// TIA Portal project "Industrial_sorter" (V17)

(* hardware
DEVICE "S7-1500/ET200MP station_1"  S7-1500 station
   slot 0: "Rail_0"  Rack  6ES7 590-1***0-0AA0
   slot 1: "PLC_1"  CPU 1511-1 PN  6ES7 511-1AK00-0AB0  V1.8
      slot 3: "CPU display_1"  6ES7591-1AA00-0AA0
      slot 32768: "PROFINET interface_1"  X1
         slot 32769: "Port_1"  X1 P1
         slot 32770: "Port_2"  X1 P2
*)

// ===== PLC "PLC_1"  CPU 1511-1 PN =====

DATA_BLOCK "Data_block_1"   // DB1
{ S7_Optimized_Access := 'FALSE' }
VERSION : 0.1
   VAR
      Nastro1_run : Bool;
      Fotocellula_ingresso_nastro1 : Bool;
      Val_induttivo : Bool;
      Val_capacitivo : Bool;
      Peso : Real;
      Fotocellula_scan : Bool;
      Fotocellula_ingresso_nastro2 : Bool;
      Tip_oggetto : Int;
      Nastro2_run : Bool;
      Pusher_avanza : Bool;
      Pusher_rientra : Bool;
      Posizione_carrello : Int;
      State_machine : Int;
      Contenitore_target : Int;
      Posizione_target_carrello : Int;
      Posizione_oggetto_X : Real;
      Posizione_oggetto_Y : Real := -1000.0;
      Timer_nastro_ET : DInt;
      Timer_nastro_PT : DInt;
      Sensore_no_oggetti : Bool := false;
      Sistema_START : Bool;
      Sistema_STOP : Bool;
      tempvar1 : Int;
      Contatore : Int;
      Allarme_generale : Bool;
      Allarme_no_tipologia : Bool;
   END_VAR
BEGIN
END_DATA_BLOCK

// folder: System blocks/Program resources

DATA_BLOCK "IEC_Timer_0_DB"   // DB2
{ S7_Optimized_Access := 'TRUE' }
AUTHOR : Simatic
FAMILY : IEC
NAME : IEC_TMR
VERSION : 1.0
// stored: InstanceOfName IEC_TIMER
"IEC_TIMER"
BEGIN
END_DATA_BLOCK

DATA_BLOCK "IEC_Timer_0_DB_1"   // DB3
{ S7_Optimized_Access := 'TRUE' }
AUTHOR : Simatic
FAMILY : IEC
NAME : IEC_TMR
VERSION : 1.0
// stored: InstanceOfName IEC_TIMER
"IEC_TIMER"
BEGIN
END_DATA_BLOCK

DATA_BLOCK "IEC_Timer_0_DB_2"   // DB4
{ S7_Optimized_Access := 'TRUE' }
AUTHOR : Simatic
FAMILY : IEC
NAME : IEC_TMR
VERSION : 1.0
// stored: InstanceOfName IEC_TIMER
"IEC_TIMER"
BEGIN
END_DATA_BLOCK

DATA_BLOCK "IEC_Timer_0_DB_3"   // DB5
{ S7_Optimized_Access := 'TRUE' }
AUTHOR : Simatic
FAMILY : IEC
NAME : IEC_TMR
VERSION : 1.0
// stored: InstanceOfName IEC_TIMER
"IEC_TIMER"
BEGIN
END_DATA_BLOCK

DATA_BLOCK "IEC_Timer_0_DB_4"   // DB6
{ S7_Optimized_Access := 'TRUE' }
AUTHOR : Simatic
FAMILY : IEC
NAME : IEC_TMR
VERSION : 1.0
// stored: InstanceOfName IEC_TIMER
"IEC_TIMER"
BEGIN
END_DATA_BLOCK

DATA_BLOCK "IEC_Timer_0_DB_5"   // DB7
{ S7_Optimized_Access := 'TRUE' }
AUTHOR : Simatic
FAMILY : IEC
NAME : IEC_TMR
VERSION : 1.0
// stored: InstanceOfName IEC_TIMER
"IEC_TIMER"
BEGIN
END_DATA_BLOCK

DATA_BLOCK "IEC_Timer_0_DB_7"   // DB11
{ S7_Optimized_Access := 'TRUE' }
AUTHOR : Simatic
FAMILY : IEC
NAME : IEC_TMR
VERSION : 1.0
// stored: InstanceOfName IEC_TIMER
"IEC_TIMER"
BEGIN
END_DATA_BLOCK

// folder: (top level)

ORGANIZATION_BLOCK "Main"   // OB1, LAD, ProgramCycle
TITLE = "Main Program Sweep (Cycle)"
{ S7_Optimized_Access := 'FALSE' }
VERSION : 0.1
   VAR_TEMP
      EV_CLASS : Byte;   // Bits 0-3 = 1:Coming event, Bits 4-7 = 1:Event class 1
      SCAN_1 : Byte;   // 1:Initial call of the OB, 3: Call 2-n of the OB
      PRIORITY : Byte;   // Priority of OB Execution
      OB_NUMBR : Byte;   // OB number
      RESERVED_1 : Byte;   // Reserved for system
      RESERVED_2 : Byte;   // Reserved for system
      PREV_CYCLE : Int;   // Previous program cycle time (milliseconds)
      MIN_CYCLE : Int;   // Minimum program cycle time (milliseconds)
      MAX_CYCLE : Int;   // Maximum program cycle time (milliseconds)
      DATE_TIME : Date_And_Time;   // Date and time OB started
   END_VAR
   VAR_TEMP   // added for the SCL form of the ladder/FBD networks
      _w1 : Bool;
      _w2 : Bool;
   END_VAR
BEGIN

REGION Network 1
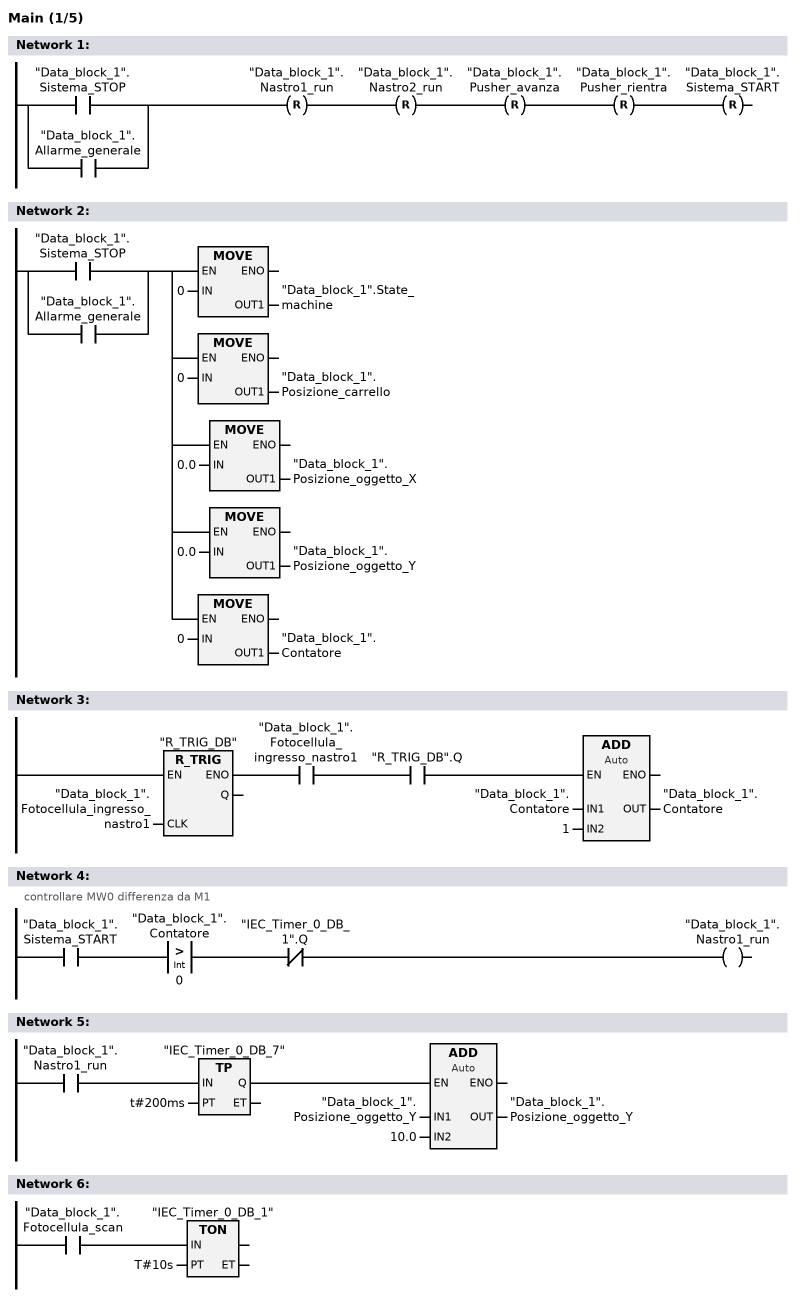
   RUNG wire#powerrail
      Contact( "Data_block_1".Sistema_STOP )
      wire#w1
      R_Coil( "Data_block_1".Nastro1_run )
      R_Coil( "Data_block_1".Nastro2_run )
      R_Coil( "Data_block_1".Pusher_avanza )
      R_Coil( "Data_block_1".Pusher_rientra )
      R_Coil( "Data_block_1".Sistema_START )
   END_RUNG
   RUNG wire#powerrail
      Contact( "Data_block_1".Allarme_generale )
   END_RUNG wire#w1
   // the same network as SCL:
   IF "Data_block_1".Sistema_STOP OR "Data_block_1".Allarme_generale THEN
       "Data_block_1".Nastro1_run := FALSE;
       "Data_block_1".Nastro2_run := FALSE;
       "Data_block_1".Pusher_avanza := FALSE;
       "Data_block_1".Pusher_rientra := FALSE;
       "Data_block_1".Sistema_START := FALSE;
   END_IF;
END_REGION

REGION Network 2
   RUNG wire#powerrail
      Contact( "Data_block_1".Sistema_STOP )
      wire#w1
      Move(in := 0, out1 => "Data_block_1".State_machine)
   END_RUNG
   RUNG wire#powerrail
      Contact( "Data_block_1".Allarme_generale )
   END_RUNG wire#w1
   RUNG wire#w1
      Move(in := 0, out1 => "Data_block_1".Posizione_carrello)
   END_RUNG
   RUNG wire#w1
      Move(in := 0.0, out1 => "Data_block_1".Posizione_oggetto_X)
   END_RUNG
   RUNG wire#w1
      Move(in := 0.0, out1 => "Data_block_1".Posizione_oggetto_Y)
   END_RUNG
   RUNG wire#w1
      Move(in := 0, out1 => "Data_block_1".Contatore)
   END_RUNG
   // the same network as SCL:
   IF "Data_block_1".Sistema_STOP OR "Data_block_1".Allarme_generale THEN
       "Data_block_1".State_machine := 0;
       "Data_block_1".Posizione_carrello := 0;
       "Data_block_1".Posizione_oggetto_X := 0.0;
       "Data_block_1".Posizione_oggetto_Y := 0.0;
       "Data_block_1".Contatore := 0;
   END_IF;
END_REGION

REGION Network 3
   // ENO of a box is taken as its EN; it also drops when the box reports an error
   "R_TRIG_DB"(CLK := "Data_block_1".Fotocellula_ingresso_nastro1);   // R_TRIG
   IF "Data_block_1".Fotocellula_ingresso_nastro1 AND "R_TRIG_DB".Q THEN
       "Data_block_1".Contatore := "Data_block_1".Contatore + 1;
   END_IF;
END_REGION

REGION Network 4
   // controllare MW0 differenza da M1
   RUNG wire#powerrail
      Contact( "Data_block_1".Sistema_START )
      { S7_Templates := "SrcType := Int" } GT_Contact(in1 := "Data_block_1".Contatore, in2 := 0)
      I_Contact( "IEC_Timer_0_DB_1".Q )
      Coil( "Data_block_1".Nastro1_run )
   END_RUNG
   // the same network as SCL:
   "Data_block_1".Nastro1_run := "Data_block_1".Sistema_START AND ("Data_block_1".Contatore > 0) AND NOT "IEC_Timer_0_DB_1".Q;
END_REGION

REGION Network 5
   "IEC_Timer_0_DB_7".TP(IN := "Data_block_1".Nastro1_run, PT := t#200ms);
   IF "IEC_Timer_0_DB_7".Q THEN
       "Data_block_1".Posizione_oggetto_Y := "Data_block_1".Posizione_oggetto_Y + 10.0;
   END_IF;
END_REGION

REGION Network 6
   "IEC_Timer_0_DB_1".TON(IN := "Data_block_1".Fotocellula_scan, PT := T#10s);
END_REGION

REGION Network 7
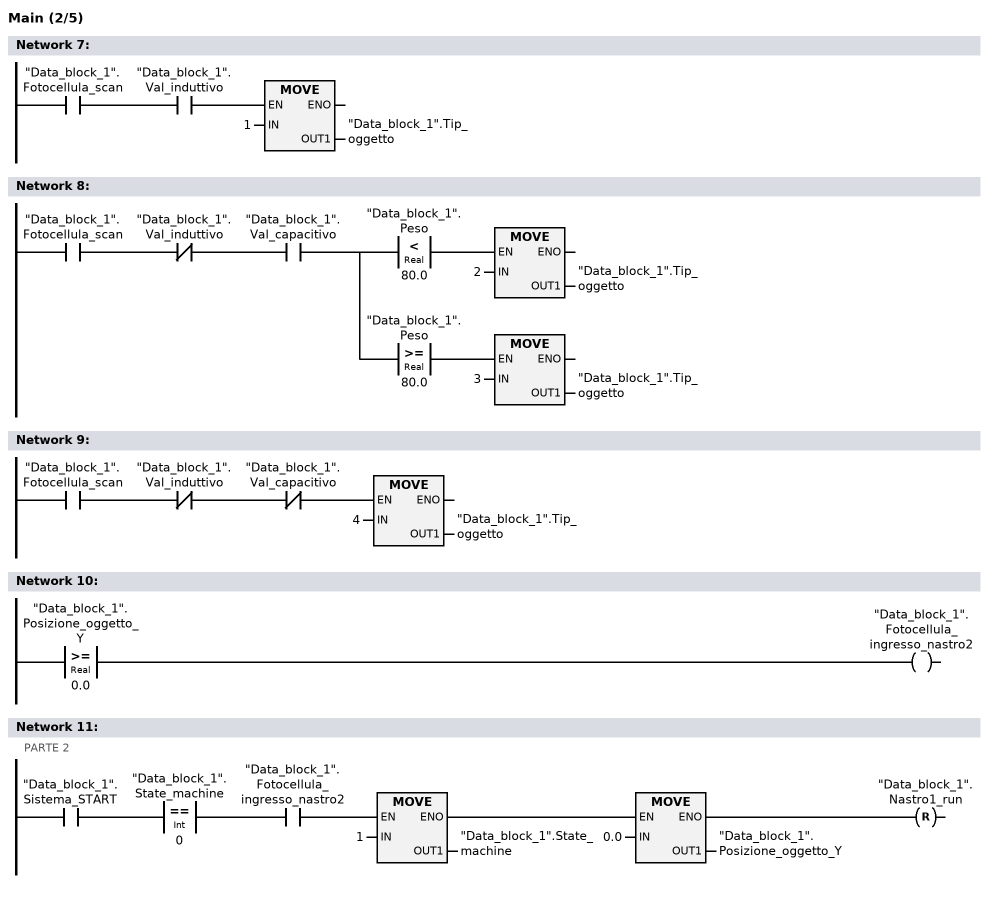
   RUNG wire#powerrail
      Contact( "Data_block_1".Fotocellula_scan )
      Contact( "Data_block_1".Val_induttivo )
      Move(in := 1, out1 => "Data_block_1".Tip_oggetto)
   END_RUNG
   // the same network as SCL:
   IF "Data_block_1".Fotocellula_scan AND "Data_block_1".Val_induttivo THEN
       "Data_block_1".Tip_oggetto := 1;
   END_IF;
END_REGION

REGION Network 8
   RUNG wire#powerrail
      Contact( "Data_block_1".Fotocellula_scan )
      I_Contact( "Data_block_1".Val_induttivo )
      Contact( "Data_block_1".Val_capacitivo )
      wire#w1
      { S7_Templates := "SrcType := Real" } LT_Contact(in1 := "Data_block_1".Peso, in2 := 80.0)
      Move(in := 2, out1 => "Data_block_1".Tip_oggetto)
   END_RUNG
   RUNG wire#w1
      { S7_Templates := "SrcType := Real" } GE_Contact(in1 := "Data_block_1".Peso, in2 := 80.0)
      Move(in := 3, out1 => "Data_block_1".Tip_oggetto)
   END_RUNG
   // the same network as SCL:
   #_w1 := "Data_block_1".Fotocellula_scan AND NOT "Data_block_1".Val_induttivo AND "Data_block_1".Val_capacitivo;
   IF #_w1 AND ("Data_block_1".Peso < 80.0) THEN "Data_block_1".Tip_oggetto := 2; END_IF;
   IF #_w1 AND ("Data_block_1".Peso >= 80.0) THEN "Data_block_1".Tip_oggetto := 3; END_IF;
END_REGION

REGION Network 9
   RUNG wire#powerrail
      Contact( "Data_block_1".Fotocellula_scan )
      I_Contact( "Data_block_1".Val_induttivo )
      I_Contact( "Data_block_1".Val_capacitivo )
      Move(in := 4, out1 => "Data_block_1".Tip_oggetto)
   END_RUNG
   // the same network as SCL:
   IF "Data_block_1".Fotocellula_scan AND NOT "Data_block_1".Val_induttivo AND NOT "Data_block_1".Val_capacitivo THEN
       "Data_block_1".Tip_oggetto := 4;
   END_IF;
END_REGION

REGION Network 10
   RUNG wire#powerrail
      { S7_Templates := "SrcType := Real" } GE_Contact(in1 := "Data_block_1".Posizione_oggetto_Y, in2 := 0.0)
      Coil( "Data_block_1".Fotocellula_ingresso_nastro2 )
   END_RUNG
   // the same network as SCL:
   "Data_block_1".Fotocellula_ingresso_nastro2 := "Data_block_1".Posizione_oggetto_Y >= 0.0;
END_REGION

REGION Network 11
   // PARTE 2
   RUNG wire#powerrail
      Contact( "Data_block_1".Sistema_START )
      { S7_Templates := "SrcType := Int" } EQ_Contact(in1 := "Data_block_1".State_machine, in2 := 0)
      Contact( "Data_block_1".Fotocellula_ingresso_nastro2 )
      Move(in := 1, out1 => "Data_block_1".State_machine)
      Move(in := 0.0, out1 => "Data_block_1".Posizione_oggetto_Y)
      R_Coil( "Data_block_1".Nastro1_run )
   END_RUNG
   // the same network as SCL:
   #_w1 := "Data_block_1".Sistema_START AND ("Data_block_1".State_machine = 0) AND "Data_block_1".Fotocellula_ingresso_nastro2;
   IF #_w1 THEN
       "Data_block_1".State_machine := 1;
       "Data_block_1".Posizione_oggetto_Y := 0.0;
       "Data_block_1".Nastro1_run := FALSE;
   END_IF;
END_REGION

REGION Network 12
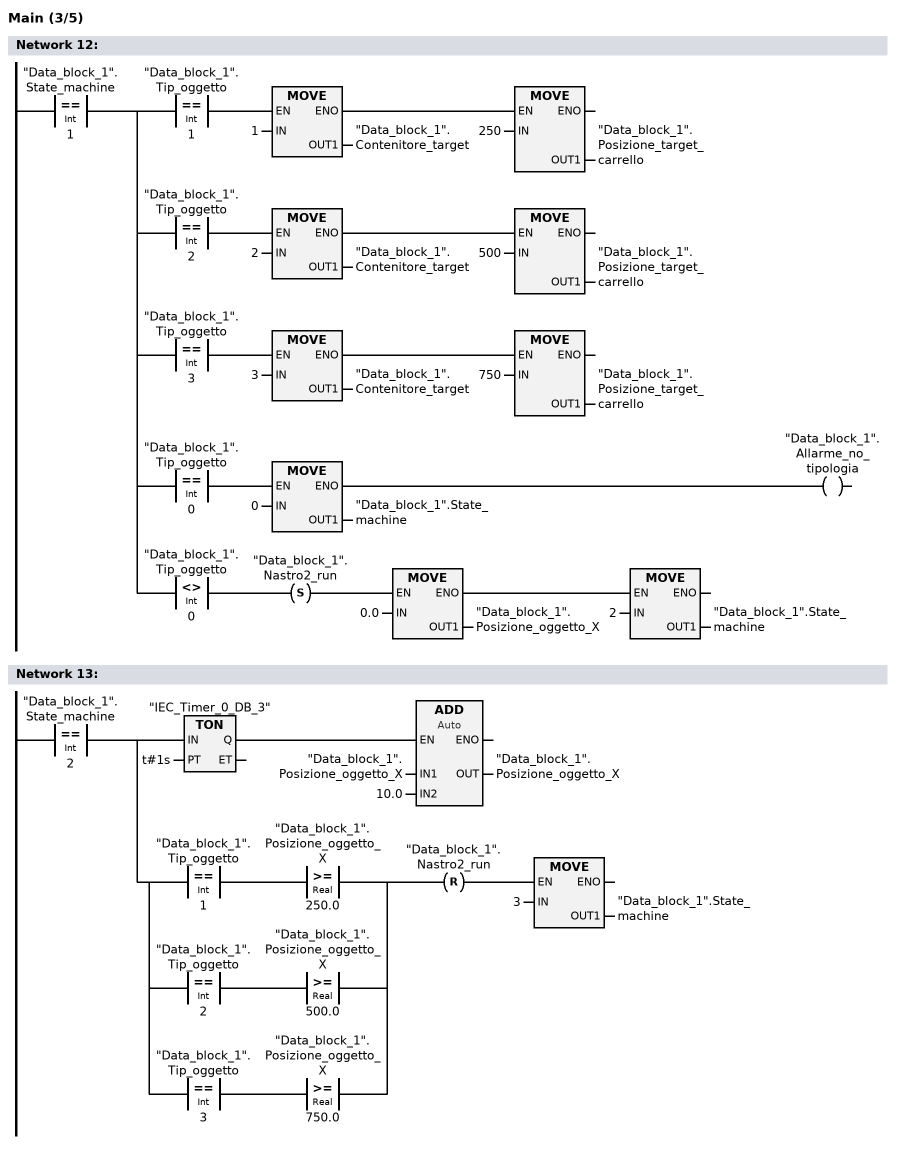
   RUNG wire#powerrail
      { S7_Templates := "SrcType := Int" } EQ_Contact(in1 := "Data_block_1".State_machine, in2 := 1)
      wire#w1
      { S7_Templates := "SrcType := Int" } EQ_Contact(in1 := "Data_block_1".Tip_oggetto, in2 := 1)
      Move(in := 1, out1 => "Data_block_1".Contenitore_target)
      Move(in := 250, out1 => "Data_block_1".Posizione_target_carrello)
   END_RUNG
   RUNG wire#w1
      { S7_Templates := "SrcType := Int" } EQ_Contact(in1 := "Data_block_1".Tip_oggetto, in2 := 2)
      Move(in := 2, out1 => "Data_block_1".Contenitore_target)
      Move(in := 500, out1 => "Data_block_1".Posizione_target_carrello)
   END_RUNG
   RUNG wire#w1
      { S7_Templates := "SrcType := Int" } EQ_Contact(in1 := "Data_block_1".Tip_oggetto, in2 := 3)
      Move(in := 3, out1 => "Data_block_1".Contenitore_target)
      Move(in := 750, out1 => "Data_block_1".Posizione_target_carrello)
   END_RUNG
   RUNG wire#w1
      { S7_Templates := "SrcType := Int" } EQ_Contact(in1 := "Data_block_1".Tip_oggetto, in2 := 0)
      Move(in := 0, out1 => "Data_block_1".State_machine)
      Coil( "Data_block_1".Allarme_no_tipologia )
   END_RUNG
   RUNG wire#w1
      { S7_Templates := "SrcType := Int" } NE_Contact(in1 := "Data_block_1".Tip_oggetto, in2 := 0)
      S_Coil( "Data_block_1".Nastro2_run )
      Move(in := 0.0, out1 => "Data_block_1".Posizione_oggetto_X)
      Move(in := 2, out1 => "Data_block_1".State_machine)
   END_RUNG
   // the same network as SCL:
   #_w1 := "Data_block_1".State_machine = 1;
   IF #_w1 AND ("Data_block_1".Tip_oggetto = 1) THEN
       "Data_block_1".Contenitore_target := 1;
       "Data_block_1".Posizione_target_carrello := 250;
   END_IF;
   IF #_w1 AND ("Data_block_1".Tip_oggetto = 2) THEN
       "Data_block_1".Contenitore_target := 2;
       "Data_block_1".Posizione_target_carrello := 500;
   END_IF;
   IF #_w1 AND ("Data_block_1".Tip_oggetto = 3) THEN
       "Data_block_1".Contenitore_target := 3;
       "Data_block_1".Posizione_target_carrello := 750;
   END_IF;
   #_w2 := #_w1 AND ("Data_block_1".Tip_oggetto = 0);
   IF #_w2 THEN "Data_block_1".State_machine := 0; END_IF;
   "Data_block_1".Allarme_no_tipologia := #_w2;
   IF #_w1 AND ("Data_block_1".Tip_oggetto <> 0) THEN
       "Data_block_1".Nastro2_run := TRUE;
       "Data_block_1".Posizione_oggetto_X := 0.0;
       "Data_block_1".State_machine := 2;
   END_IF;
END_REGION

REGION Network 13
   #_w1 := "Data_block_1".State_machine = 2;
   "IEC_Timer_0_DB_3".TON(IN := #_w1, PT := t#1s);
   IF "IEC_Timer_0_DB_3".Q THEN
       "Data_block_1".Posizione_oggetto_X := "Data_block_1".Posizione_oggetto_X + 10.0;
   END_IF;
   IF #_w1 AND ((("Data_block_1".Tip_oggetto = 1) AND ("Data_block_1".Posizione_oggetto_X >= 250.0)) OR (("Data_block_1".Tip_oggetto = 2) AND ("Data_block_1".Posizione_oggetto_X >= 500.0)) OR (("Data_block_1".Tip_oggetto = 3) AND ("Data_block_1".Posizione_oggetto_X >= 750.0))) THEN
       "Data_block_1".Nastro2_run := FALSE;
       "Data_block_1".State_machine := 3;
   END_IF;
END_REGION

REGION Network 14
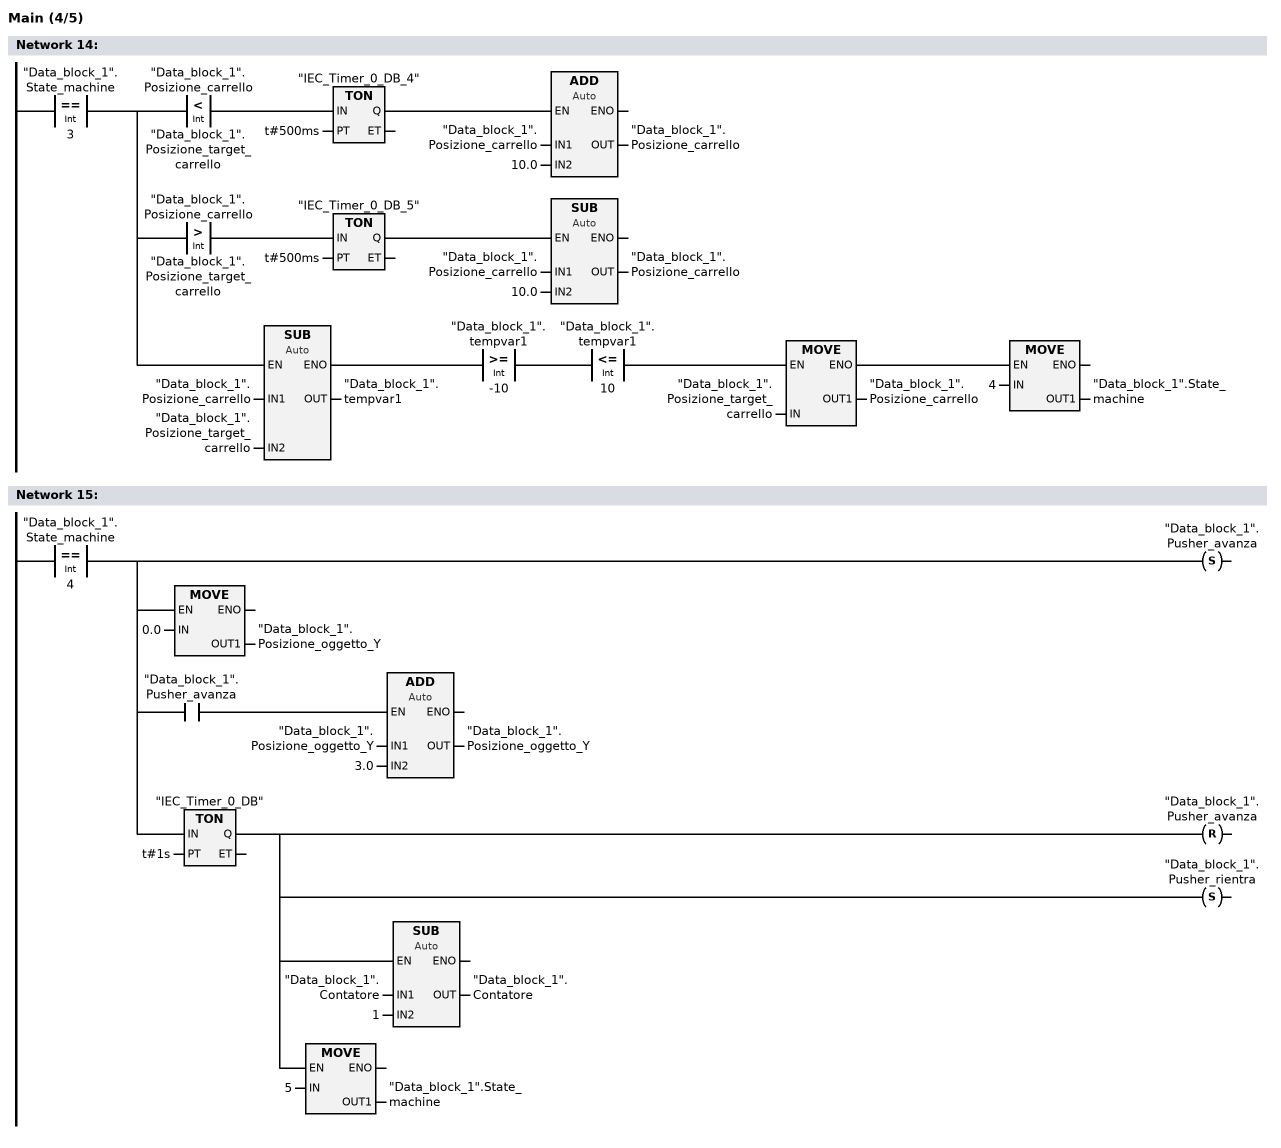
   #_w1 := "Data_block_1".State_machine = 3;
   "IEC_Timer_0_DB_4".TON(IN := #_w1 AND ("Data_block_1".Posizione_carrello < "Data_block_1".Posizione_target_carrello),
                          PT := t#500ms);
   IF "IEC_Timer_0_DB_4".Q THEN
       "Data_block_1".Posizione_carrello := "Data_block_1".Posizione_carrello + 10.0;
   END_IF;
   "IEC_Timer_0_DB_5".TON(IN := #_w1 AND ("Data_block_1".Posizione_carrello > "Data_block_1".Posizione_target_carrello),
                          PT := t#500ms);
   IF "IEC_Timer_0_DB_5".Q THEN
       "Data_block_1".Posizione_carrello := "Data_block_1".Posizione_carrello - 10.0;
   END_IF;
   IF #_w1 THEN
       "Data_block_1".tempvar1 := "Data_block_1".Posizione_carrello - "Data_block_1".Posizione_target_carrello;
   END_IF;
   IF #_w1 AND ("Data_block_1".tempvar1 >= (-10)) AND ("Data_block_1".tempvar1 <= 10) THEN
       "Data_block_1".Posizione_carrello := "Data_block_1".Posizione_target_carrello;
       "Data_block_1".State_machine := 4;
   END_IF;
END_REGION

REGION Network 15
   #_w1 := "Data_block_1".State_machine = 4;
   IF #_w1 THEN
       "Data_block_1".Pusher_avanza := TRUE;
       "Data_block_1".Posizione_oggetto_Y := 0.0;
   END_IF;
   IF #_w1 AND "Data_block_1".Pusher_avanza THEN
       "Data_block_1".Posizione_oggetto_Y := "Data_block_1".Posizione_oggetto_Y + 3.0;
   END_IF;
   "IEC_Timer_0_DB".TON(IN := #_w1, PT := t#1s);
   IF "IEC_Timer_0_DB".Q THEN
       "Data_block_1".Pusher_avanza := FALSE;
       "Data_block_1".Pusher_rientra := TRUE;
       "Data_block_1".Contatore := "Data_block_1".Contatore - 1;
       "Data_block_1".State_machine := 5;
   END_IF;
END_REGION

REGION Network 16
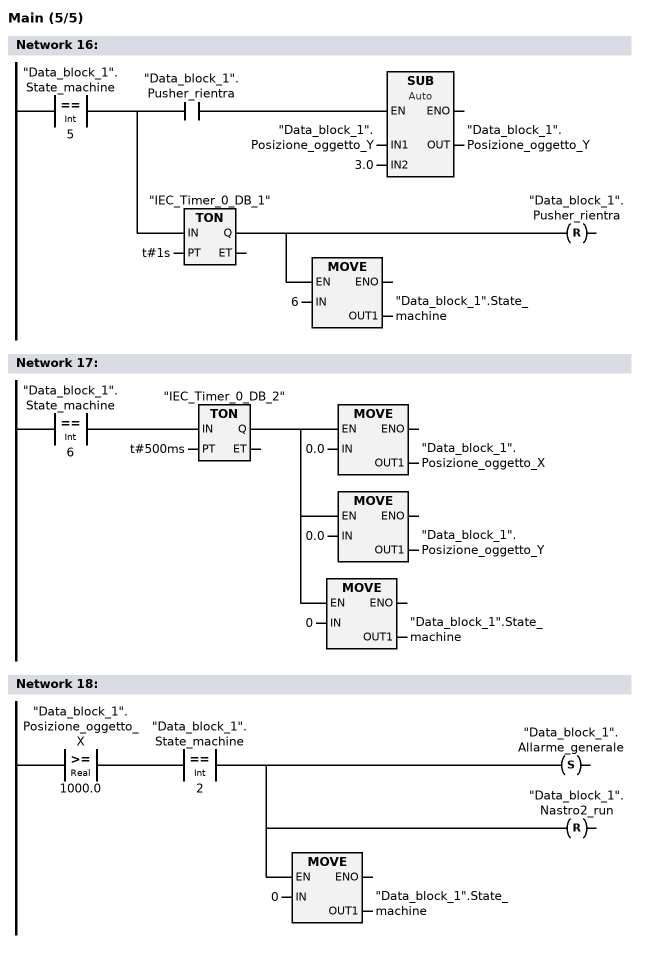
   #_w1 := "Data_block_1".State_machine = 5;
   IF #_w1 AND "Data_block_1".Pusher_rientra THEN
       "Data_block_1".Posizione_oggetto_Y := "Data_block_1".Posizione_oggetto_Y - 3.0;
   END_IF;
   "IEC_Timer_0_DB_1".TON(IN := #_w1, PT := t#1s);
   IF "IEC_Timer_0_DB_1".Q THEN
       "Data_block_1".Pusher_rientra := FALSE;
       "Data_block_1".State_machine := 6;
   END_IF;
END_REGION

REGION Network 17
   "IEC_Timer_0_DB_2".TON(IN := "Data_block_1".State_machine = 6, PT := t#500ms);
   IF "IEC_Timer_0_DB_2".Q THEN
       "Data_block_1".Posizione_oggetto_X := 0.0;
       "Data_block_1".Posizione_oggetto_Y := 0.0;
       "Data_block_1".State_machine := 0;
   END_IF;
END_REGION

REGION Network 18
   RUNG wire#powerrail
      { S7_Templates := "SrcType := Real" } GE_Contact(in1 := "Data_block_1".Posizione_oggetto_X, in2 := 1000.0)
      { S7_Templates := "SrcType := Int" } EQ_Contact(in1 := "Data_block_1".State_machine, in2 := 2)
      wire#w1
      S_Coil( "Data_block_1".Allarme_generale )
   END_RUNG
   RUNG wire#w1
      R_Coil( "Data_block_1".Nastro2_run )
   END_RUNG
   RUNG wire#w1
      Move(in := 0, out1 => "Data_block_1".State_machine)
   END_RUNG
   // the same network as SCL:
   IF ("Data_block_1".Posizione_oggetto_X >= 1000.0) AND ("Data_block_1".State_machine = 2) THEN
       "Data_block_1".Allarme_generale := TRUE;
       "Data_block_1".Nastro2_run := FALSE;
       "Data_block_1".State_machine := 0;
   END_IF;
END_REGION
END_ORGANIZATION_BLOCK